(* PLC project logical_or, Dassault Systèmes ControlBuild 2024x *)
(* stored: creationDateTime 2023-10-03T11:13:28-01:00 *)

(* This module makes a "logical OR" operation between two inputs. Result is a boolean. *)
FUNCTION_BLOCK equipment_library.logical_or
  VAR_INPUT
    inputBit1 : BOOL := false;
    inputBit2 : BOOL := false;
  END_VAR
  VAR_OUTPUT
    outputBit : BOOL := false;
  END_VAR
  VAR CONSTANT
    input1Logic : BOOL := true;
    input2Logic : BOOL := true;
    outputLogic : BOOL := true;
  END_VAR
  VAR
    d_output : BOOL := false;
    v_d_output : BOOL := true;
  END_VAR


ACTION C_source_code:
/* ----------------------------------------------------------------	*/
/* Type : Model of Operative Behaviour					*/
/* Category :  Toolbox							*/
/* Author : Dassault Systemes						*/
/* Update date : June 2018						*/
/* ----------------------------------------------------------------	*/
/* This module makes a "logical OR" operation between two inputs.	*/
/* Result is a boolean.							*/
/* The output can be preset	by the user					*/
/* ----------------------------------------------------------------	*/

if (d_output) outputBit = v_d_output;
else
	outputBit = ((inputBit1 ^ ! input1Logic) | (inputBit2 ^ ! input2Logic)) ^ ! outputLogic;
END_ACTION
END_FUNCTION_BLOCK
